(*

short summary
=============

.. <legal notes>

legal notes
=================
| SPDX-FileCopyrightText: © 2023 ekvip automation GmbH <info@ekvip.de>
| SPDX-License-Identifier: Apache-2.0
| For details check: Apache-2.0_

.. _Apache-2.0: https://www.apache.org/licenses/LICENSE-2.0

.. </legal notes>

enumeration values
==================

*)

{warning 'header is generated please add your documentation'}
{attribute 'qualified_only'}
{attribute 'strict'}
TYPE TypeToTest :
(
	TEST_STRING 	:= 0,
	TEST_WSTRING 	:= 1
);
END_TYPE

(* stored: Version 1.1.0.1, ProductVersion 3.1.4024.12
   DUT TypeToTest: Id {89460358-64bd-4d98-8d84-50ae4ad08ecf} *)
